// SIMATIC STEP 7 (V5.x) project star_delta_starting
// CPU: CPU 317-2 DP
// station: Hardware
// station: SIMATIC 300(1)
// station: P_ADR_BUS
// program: Programa S7(1)

SYMBOL_TABLE
"Motor_starting_db"	DB 1	FB 1
"Motor_starting"	FB 1	FB 1
"START_PB"	I 0.0	BOOL	// Start Pushbutton o Motor Start Command
"MOTOR_PROTECTION"	I 0.1	BOOL	// Motor Protection Circuit Breaker (MPCB)
"E_STOP"	I 0.2	BOOL	// Emergency Stop (E-Stop)
"Cycle Execution"	OB 1	OB 1
"MAIN_CONTACTOR"	Q 4.0	BOOL	// Main Motor Contactor
"STAR_CONTACTOR"	Q 4.1	BOOL	// Star Contactor
"DELTA_CONTACTOR"	Q 4.2	BOOL	// Delta Contactor
"RUN_LAMP"	Q 4.3	BOOL	// Run Indicator Lamp
"KT"	T 0	TIMER	// Start-up Time
END_SYMBOL_TABLE

FUNCTION_BLOCK "Motor_starting"	// FB 1
VERSION : 0.1
VAR_INPUT
  START : BOOL ;
  STOP : BOOL ;
  CIRCUIT_BREAKER : BOOL ;
  TIMER_KT : TIMER ;
  TIMER_DURATION : S5TIME ;
END_VAR
VAR_OUTPUT
  KM1_MAIN : BOOL ;
  KM2_STAR : BOOL ;
  KM3_DELTA : BOOL ;
  LAMP : BOOL ;
END_VAR
BEGIN
NETWORK
TITLE = Motor starting sequence
      A(;
      O     #START;
      O     #KM1_MAIN;
      );
      AN    #CIRCUIT_BREAKER;
      A     #STOP;
      =     L 0.0;
      A     L 0.0;
      BLD   102;
      =     #KM1_MAIN;
      A     L 0.0;
      BLD   102;
      =     #LAMP;
      A     L 0.0;
      L     #TIMER_DURATION;
      T     LD 1;
      TAK;
      T     LD 5;
      L     #TIMER_KT;
      T     LW 9;
      L     LD 5;
      L     LD 1;
      SD    T [LW 9];
      NOP   0;
      NOP   0;
      NOP   0;
      NOP   0;
NETWORK
TITLE = Star sequence
      A     #KM1_MAIN;
      AN    #KM3_DELTA;
      T     LD 0;
      TAK;
      T     LD 4;
      L     #TIMER_KT;
      T     LW 8;
      L     LD 4;
      L     LD 0;
      AN    T [LW 8];
      =     #KM2_STAR;
NETWORK
TITLE = Delta sequence
      A     #KM1_MAIN;
      AN    #KM2_STAR;
      T     LD 0;
      TAK;
      T     LD 4;
      L     #TIMER_KT;
      T     LW 8;
      L     LD 4;
      L     LD 0;
      A     T [LW 8];
      =     #KM3_DELTA;
END_FUNCTION_BLOCK

DATA_BLOCK "Motor_starting_db"	// DB 1
VERSION : 0.1
"Motor_starting"
BEGIN
END_DATA_BLOCK

ORGANIZATION_BLOCK "Cycle Execution"	// OB 1
TITLE = "Main Program Sweep (Cycle)"
VERSION : 0.1
VAR_TEMP
  OB1_EV_CLASS : BYTE ;	//Bits 0-3 = 1 (Coming event), Bits 4-7 = 1 (Event class 1)
  OB1_SCAN_1 : BYTE ;	//1 (Cold restart scan 1 of OB 1), 3 (Scan 2-n of OB 1)
  OB1_PRIORITY : BYTE ;	//Priority of OB Execution
  OB1_OB_NUMBR : BYTE ;	//1 (Organization block 1, OB1)
  OB1_RESERVED_1 : BYTE ;	//Reserved for system
  OB1_RESERVED_2 : BYTE ;	//Reserved for system
  OB1_PREV_CYCLE : INT ;	//Cycle time of previous OB1 scan (milliseconds)
  OB1_MIN_CYCLE : INT ;	//Minimum cycle time of OB1 (milliseconds)
  OB1_MAX_CYCLE : INT ;	//Maximum cycle time of OB1 (milliseconds)
  OB1_DATE_TIME : DATE_AND_TIME ;	//Date and time OB1 started
END_VAR
BEGIN
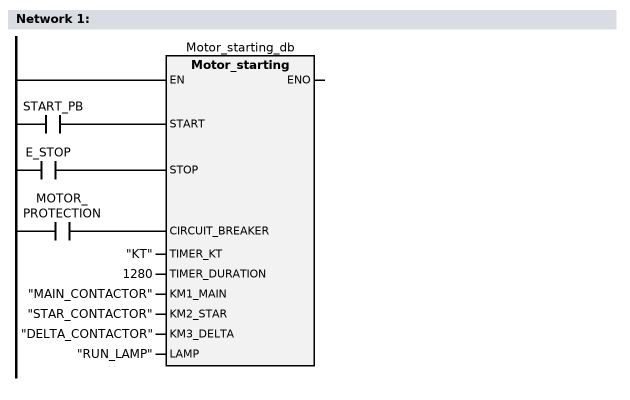
NETWORK
TITLE =
      A     "START_PB";
      =     L 20.0;
      BLD   103;
      A     "E_STOP";
      =     L 20.1;
      BLD   103;
      A     "MOTOR_PROTECTION";
      =     L 20.2;
      BLD   103;
      CALL  "Motor_starting" , "Motor_starting_db" (
           START                    := L 20.0,
           STOP                     := L 20.1,
           CIRCUIT_BREAKER          := L 20.2,
           TIMER_KT                 := "KT",
           TIMER_DURATION           := 1280,
           KM1_MAIN                 := "MAIN_CONTACTOR",
           KM2_STAR                 := "STAR_CONTACTOR",
           KM3_DELTA                := "DELTA_CONTACTOR",
           LAMP                     := "RUN_LAMP");
      NOP   0;
END_ORGANIZATION_BLOCK
